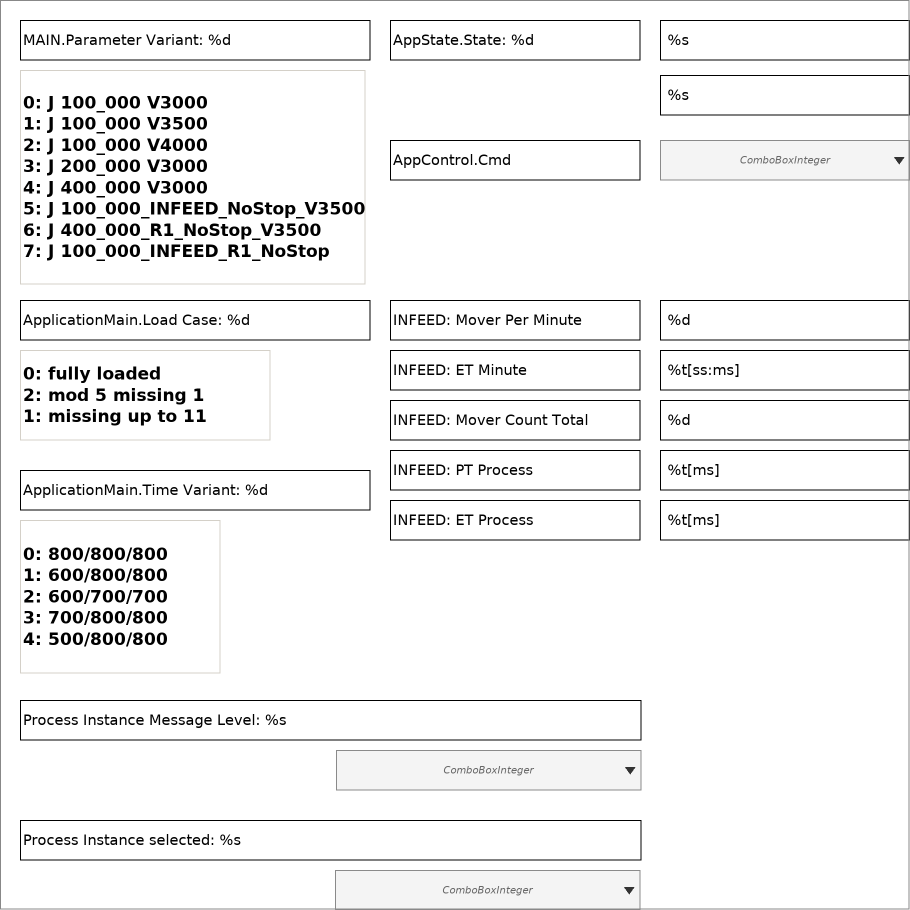
VISUALIZATION SIM_TEST  // 910x910
    Rectangle (20,300 350x40), "ApplicationMain.Load Case: %d", text variable: GVL_APPLICATION.ApplicationMain._nLoadCase
        OnMouseClick: write the text variable via VisuDialogs.Numpad, min 0, max 2
    Rectangle (20,470 350x40), "ApplicationMain.Time Variant: %d", text variable: GVL_APPLICATION.ApplicationMain._nTimeVariant
        OnMouseClick: write the text variable via VisuDialogs.Numpad, min 0, max 100
    Rectangle (20,20 350x40), "MAIN.Parameter Variant: %d", text variable: MAIN.nParameterVariant
        OnMouseClick: write the text variable via VisuDialogs.Numpad, min 0, max 100
    Textfield (20,520 200x153), "0: 800/800/800 1: 600/800/800 2: 600/700/700 3: 700/800/800 4: 500/800/800"
    Textfield (20,350 250x90), "0: fully loaded 2: mod 5 missing 1 1: missing up to 11"
    Textfield (20,70 345x214), "0: J 100_000 V3000 1: J 100_000 V3500 2: J 100_000 V4000 3: J 200_000 V3000 4: J 400_000 V3000 5: J 100_000_INFEED_NoStop_V3500 6: J 400_000_R1_NoStop_V3500 7: J 100_000_INFEED_R1_NoStop"
    Rectangle (390,140 250x40), "AppControl.Cmd"
    ComboBoxInteger (660,140 250x40), variable: GVL_APPLICATION.AppControl.Cmd, text list: 'TL_E_INSTANCE_CMD'
    Rectangle (390,20 250x40), "AppState.State: %d", text variable: GVL_APPLICATION.AppState.AppState
    Rectangle (660,75 250x40), "%s", text variable: GVL_APPLICATION.ApplicationMain._sAppResult
    Rectangle (390,300 250x40), "INFEED: Mover Per Minute"
    Rectangle (660,300 250x40), "%d", text variable: GVL_APPLICATION.ProcessCollector[2]._AllStationMoverPerMinute
    Rectangle (390,400 250x40), "INFEED: Mover Count Total"
    Rectangle (660,400 250x40), "%d", text variable: GVL_APPLICATION.ProcessCollector[2]._nMoverCountTotal
    Rectangle (390,500 250x40), "INFEED: ET Process"
    Rectangle (660,500 250x40), "%t[ms]", text variable: GVL_APPLICATION.ApplicationMain._tonProcess[2].ET
    Rectangle (390,450 250x40), "INFEED: PT Process"
    Rectangle (660,450 250x40), "%t[ms]", text variable: GVL_APPLICATION.ApplicationMain._tProcess[2]
    Rectangle (390,350 250x40), "INFEED: ET Minute"
    Rectangle (660,350 250x40), "%t[ss:ms]", text variable: ProcessCollector[2]._tonPartsPerMinute.ET
    Rectangle (660,20 250x40), "%s", text variable: GVL_APPLICATION.ApplicationMain._sAppState
    Rectangle (20,700 621x40), "Process Instance Message Level: %s", text variable: MessageData.sMessageLevelSelected
    ComboBoxInteger (335,870 305x40), variable: MessageData.nProcessSelected, text list: 'TL_E_INSTANCE'
    ComboBoxInteger (336,750 305x40), variable: GVL_MSG.MessageLevelProcess[MessageData.nProcessSelected], text list: 'TL_E_MESSAGETYPE'
    Rectangle (20,820 621x40), "Process Instance selected: %s", text variable: MessageData.sProcessSelected
END_VISUALIZATION

(* stored: Version 1.1.0.1, ProductVersion 3.1.4024.15
   Visu SIM_TEST: Id {986ae958-2a9d-4eb4-9e8a-0f993c444b4f} *)
